FUNCTION_BLOCK FB_Candle
VAR_INPUT
END_VAR
VAR_OUTPUT
END_VAR
VAR
	dia			: REAL;
	height 		: REAL;
	numWicks 	: INT;
	weight 		: REAL;
END_VAR

END_FUNCTION_BLOCK

(* stored: Version 1.1.0.1, ProductVersion 3.1.4024.12
   POU FB_Candle: Id {06c667fb-2378-4630-8022-0be5e9be0cd6}, SpecialFunc None *)
